{attribute 'GeneratedUsingTerminal: EL6201-0000-0017'}
{attribute addProperty BoxType "EL6201-0000-0017"}
{attribute addProperty Id "Slave_11A_DO0BOOL1Slave_11A_DO1BOOL1Slave_11A_DO2BOOL1Slave_11A_DO3BOOL1Slave_11B_DO0BOOL1Slave_11B_DO1BOOL1Slave_11B_DO2BOOL1Slave_11B_DO3BOOL1"}
{attribute addProperty CRC "3699129888"}
{attribute addProperty Size "8"}
TYPE Slave_11_Outputs_DC7C3E20 :
STRUCT
	{attribute addProperty Name "Slave_11A_DO0"}
	Slave_11A_DO0 : BOOL;
	{attribute addProperty Name "Slave_11A_DO1"}
	Slave_11A_DO1 : BOOL;
	{attribute addProperty Name "Slave_11A_DO2"}
	Slave_11A_DO2 : BOOL;
	{attribute addProperty Name "Slave_11A_DO3"}
	Slave_11A_DO3 : BOOL;
	{attribute addProperty Name "Slave_11B_DO0"}
	Slave_11B_DO0 : BOOL;
	{attribute addProperty Name "Slave_11B_DO1"}
	Slave_11B_DO1 : BOOL;
	{attribute addProperty Name "Slave_11B_DO2"}
	Slave_11B_DO2 : BOOL;
	{attribute addProperty Name "Slave_11B_DO3"}
	Slave_11B_DO3 : BOOL;
END_STRUCT
END_TYPE

(* stored: Version 1.2.0.0, ProductVersion 3.1.4024.9
   DUT Slave_11_Outputs_DC7C3E20: Id {328e244e-bb7c-4cfa-baea-c144994d6c66} *)
